FUNCTION_BLOCK FB_EventLog
VAR_INPUT
	Trigger:		BOOL;
	// ADSLOG_MSGTYPE_HINT or ADSLOG_MSGTYPE_WARN or ADSLOG_MSGTYPE_ERROR
	Level:			UDINT := ADSLOG_MSGTYPE_HINT;
	FormatString: 	STRING(255) := '%s';
	OnMessage: 		STRING(255) := '';
	OffMessage:		STRING(255) := '';
	OffLevel:		UDINT := ADSLOG_MSGTYPE_HINT;
END_VAR
VAR_OUTPUT
END_VAR
VAR
	LogonTrigger: R_TRIG;
	LogoffTrigger: F_TRIG;
END_VAR

LogonTrigger(CLK := Trigger);
LogoffTrigger(CLK := Trigger);
// in case the OffLevel is not set use the default Level Value
IF OffLevel = 0 THEN
	OffLevel := Level;
END_IF
IF LogonTrigger.Q AND LEN(OnMessage)>0 THEN
	ADSLOGSTR( Level OR ADSLOG_MSGTYPE_LOG, FormatString, OnMessage);
END_IF

IF LogoffTrigger.Q AND LEN(OffMessage)>0 THEN
	ADSLOGSTR( OffLevel OR ADSLOG_MSGTYPE_LOG, FormatString, OffMessage);
END_IF

END_FUNCTION_BLOCK

(* stored: Version 1.1.0.1, ProductVersion 3.1.4024.9
   POU FB_EventLog: Id {3524ed80-3787-4549-a84e-d995fc3a40dc}, SpecialFunc None *)
